# B&R Automation Studio project AcpTrakDemoTemplate (part 2)

#### Main.st
```iecst
(*********************************************************************************
 * Copyright: 	B&R Industrial Automation GmbH
 * Author:    	B&R ES
 * Created:   	April 8, 2022/10:54 AM
 * Description:	All the shuttles crossing this process point will be unsynched.
 * Mandatory: 	NO
 *********************************************************************************)
PROGRAM _INIT

	(*******************************************************************)
	(******************* Process Configuration *************************)
	(*******************************************************************)
	PPAdr 	:= ADR(PP_Test); 	// <-- NAME A VALID PROCESS POINT
	(*** Define in/out speed & acceleration for this process ***)
	// OUT
	Speed_OUT ACCESS ADR(gSpeedEmpty); 	// <-- Bind it to Empty / Full speed global variable
	Acc_OUT	ACCESS ADR(gAccEmpty); 		// <-- Bind it to Empty / Full acceleration global variable
	(*** SceneViewer - Shuttle color after process ***)
	Red	  := 1.0;
	Green := 1.0;
	Blue  := 1.0;
	(********************************************************************)

	(* Local variable to enable/disable the process *)
	CmdEnableProcess := TRUE;
	(* Processpointreference for Functionblocks *)
	MC_BR_TrgPointEnable_AcpTrak_0.ProcessPoint 	:= PPAdr; // <-- NAME A VALID PROCESS POINT
	MC_BR_TrgPointGetInfo_AcpTrak_0.ProcessPoint 	:= PPAdr;	// <-- NAME A VALID PROCESS POINT

END_PROGRAM

PROGRAM _CYCLIC

	//////////////////// HIGH PRIORITY ///////////////////
	IF gTrakAsm.StatusDisabled THEN
		Step 		:= CHECK_TRIGGER;
	END_IF
	//////////////////////////////////////////////////////

	CASE Step OF

		CHECK_TRIGGER:

			(* When the process is enabled and the assembly is ready, the process will be activated *)
			IF((CmdEnableProcess) AND (gTrakAsm.StatusReady))THEN
				MC_BR_TrgPointEnable_AcpTrak_0.Enable := TRUE;
				(* If a shuttle passes the triggerpoint then get the axis reference *)
				IF((MC_BR_TrgPointEnable_AcpTrak_0.Valid) AND (MC_BR_TrgPointEnable_AcpTrak_0.EventCount > 0))THEN
					MC_BR_TrgPointGetInfo_AcpTrak_0.Execute := TRUE;
				END_IF
			ELSE
				(* Else the processpoint will be disabled *)
				MC_BR_TrgPointEnable_AcpTrak_0.Enable := FALSE;
			END_IF

			(* If axis reference is available, save it and go to the next step *)
			IF EDGEPOS(MC_BR_TrgPointGetInfo_AcpTrak_0.Done) THEN
			(* Save axis reference in local variable for use in step machine *)
				ShuttleAxis	:= MC_BR_TrgPointGetInfo_AcpTrak_0.TrgPointInfo.Axis;
				Step 		:= GET_USERDATA;
			END_IF

		GET_USERDATA:

			(* The userdata is copied on a local variable *)
			MC_BR_ShCopyUserData_AcpTrak_0.Axis 		:= ADR(ShuttleAxis);
			MC_BR_ShCopyUserData_AcpTrak_0.Execute 		:= TRUE;
			MC_BR_ShCopyUserData_AcpTrak_0.DataAddress	:= ADR(ShuttleUserData);
			MC_BR_ShCopyUserData_AcpTrak_0.DataSize 	:= SIZEOF(ShuttleUserData);
			MC_BR_ShCopyUserData_AcpTrak_0.Mode 		:= mcACPTRAK_USERDATA_GET;
			(* After copying go to the next step *)
			IF EDGEPOS(MC_BR_ShCopyUserData_AcpTrak_0.Done) THEN
				IF ShuttleUserData.InitDone THEN
					Step := SET_USERDATA;
				ELSE
					Step := CHECK_TRIGGER;
				END_IF
			END_IF

		SET_USERDATA:

			(* Change color to know that shuttles are in unsync. *)
			ShuttleUserData.SceneColorRed 	:= Red;
			ShuttleUserData.SceneColorGreen := Green;
			ShuttleUserData.SceneColorBlue	:= Blue;

			(* The modified userdata will be copied back on the shuttle *)
			MC_BR_ShCopyUserData_AcpTrak_0.Axis 		:= ADR(ShuttleAxis);
			MC_BR_ShCopyUserData_AcpTrak_0.Execute 		:= TRUE;
			MC_BR_ShCopyUserData_AcpTrak_0.DataAddress	:= ADR(ShuttleUserData);
			MC_BR_ShCopyUserData_AcpTrak_0.DataSize 	:= SIZEOF(ShuttleUserData);
			MC_BR_ShCopyUserData_AcpTrak_0.Mode 		:= mcACPTRAK_USERDATA_SET;
			Step := SET_USERDATA_WAIT;

		SET_USERDATA_WAIT:

			IF (MC_BR_ShCopyUserData_AcpTrak_0.Done) THEN
				Step := GO_TO_NEXT_STATION;
			END_IF

		GO_TO_NEXT_STATION:

			MC_BR_ElasticMoveVel_AcpTrak_0.Axis 	:= ADR(ShuttleAxis);
			MC_BR_ElasticMoveVel_AcpTrak_0.Execute	:= TRUE;

			Step := CHECK_TRIGGER;

	END_CASE

	(*** Call all function blocks ***)
	// MC_BR_TrgPointEnable_AcpTrak
	MC_BR_TrgPointEnable_AcpTrak_0();
	// MC_BR_TrgPointGetInfo_AcpTrak
	MC_BR_TrgPointGetInfo_AcpTrak_0();
	MC_BR_TrgPointGetInfo_AcpTrak_0.Execute  := FALSE;
	// MC_BR_ShCopyUserData_AcpTrak
	MC_BR_ShCopyUserData_AcpTrak_0();
	MC_BR_ShCopyUserData_AcpTrak_0.Execute 	 := FALSE;
	//MC_BR_ElasticMoveVel_AcpTrak_0
	MC_BR_ElasticMoveVel_AcpTrak_0.Velocity		:= Speed_OUT;
	MC_BR_ElasticMoveVel_AcpTrak_0.Acceleration	:= Acc_OUT;
	MC_BR_ElasticMoveVel_AcpTrak_0.Deceleration	:= Acc_OUT;
	MC_BR_ElasticMoveVel_AcpTrak_0.Direction	:= mcDIR_POSITIVE;
	MC_BR_ElasticMoveVel_AcpTrak_0();
	MC_BR_ElasticMoveVel_AcpTrak_0.Execute		:= FALSE;

END_PROGRAM
```

### Program Logical/Source/ProcessTemplate/PairedSh/ProcStop_P1 (IEC) - trak process - 1 pair of shuttles wait predefined time

#### Types.typ
```iecst
(*enum*)

TYPE
	StepEnum :
		(
		CHECK_TRIGGER,
		GET_SHUTTLE_DATA,
		GET_SHUTTLE_DATA_WAIT,
		GO_TO_PROCESS_STATION,
		GO_TO_PROCESS_STATION_WAIT,
		WAIT,
		SET_SHUTTLE_DATA,
		SET_SHUTTLE_DATA_WAIT,
		GO_TO_NEXT_STATION
		);
END_TYPE
```

#### Variables.var
```iecst
(*process configuration*)
VAR
	PPAdr : UDINT;
	SecAdr : UDINT;
END_VAR
(*commands*)
VAR
	CmdEnableProcess : BOOL;
END_VAR
(*sequence control*)
VAR
	Step : StepEnum;
	ShuttleAxis : ARRAY[1..2] OF McAxisType;
	ShuttleUserData : ARRAY[1..2] OF TrakShuttleUserDataType;
	WaitTime : UDINT := 500;
	ProcPointPos : LREAL;
	CntShuttle : USINT;
	ReleaseSts : BOOL;
END_VAR
(*colour configuration*)
VAR
	Red : REAL;
	Green : REAL;
	Blue : REAL;
END_VAR
(*movement configuration*)
VAR
	Speed_IN : REFERENCE TO REAL;
	Acc_IN : REFERENCE TO REAL;
	Speed_OUT : REFERENCE TO REAL;
	Acc_OUT : REFERENCE TO REAL;
END_VAR
(*FUB*)
VAR
	MC_BR_AsmReadStatus_AcpTrak_0 : MC_BR_AsmReadStatus_AcpTrak;
	MC_BR_TrgPointEnable_AcpTrak_0 : MC_BR_TrgPointEnable_AcpTrak;
	MC_BR_TrgPointGetInfo_AcpTrak_0 : MC_BR_TrgPointGetInfo_AcpTrak;
	MC_BR_ShCopyUserData_AcpTrak_0 : MC_BR_ShCopyUserData_AcpTrak;
	MC_BR_RoutedMoveAbs_AcpTrak_0 : MC_BR_RoutedMoveAbs_AcpTrak;
	MC_BR_ElasticMoveVel_AcpTrak_0 : MC_BR_ElasticMoveVel_AcpTrak;
	MC_BR_ProcPointGetInfo_AcpTrak_0 : MC_BR_ProcPointGetInfo_AcpTrak;
	TON_0 : TON;
END_VAR
```

#### Main.st
```iecst
(*********************************************************************************
 * Copyright: 	B&R Industrial Automation GmbH
 * Author:    	B&R ES
 * Created:   	April 8, 2022/10:54 AM
 * Description:	One pair of coupled shuttles will be stopped a predefined time in the
				process	station.
 * Mandatory: 	NO
 *********************************************************************************)
PROGRAM _INIT

	(*******************************************************************)
	(******************* Process Configuration *************************)
	(*******************************************************************)
	PPAdr 	:= ADR(PP_Test); 		// <-- NAME A VALID PROCESS POINT
	SecAdr	:= ADR(SectorTrackA);	// <-- NAME A VALID SECTOR
	(*** Define in/out speed & acceleration for this process ***)
	// IN
	Speed_IN ACCESS	ADR(gSpeedEmpty); 	// <-- Bind it to Empty / Full speed global variable
	Acc_IN ACCESS ADR(gAccEmpty); 		// <-- Bind it to Empty / Full acceleration global variable
	// OUT
	Speed_OUT ACCESS ADR(gSpeedFull); 	// <-- Bind it to Empty / Full speed global variable
	Acc_OUT	ACCESS ADR(gAccFull); 		// <-- Bind it to Empty / Full acceleration global variable
	(*** Define Wait Time (ms) ***)
	WaitTime := 500;
	(*** Define if it is a release station ***)
	ReleaseSts := FALSE;
	(*** SceneViewer - Shuttle color after process ***)
	Red	  := 0.02;
	Green := 0.77;
	Blue  := 0.21;
	(********************************************************************)

	CmdEnableProcess 	:= TRUE;
	Step 				:= CHECK_TRIGGER;

	MC_BR_ProcPointGetInfo_AcpTrak_0.ProcessPoint   := PPAdr;
	MC_BR_ProcPointGetInfo_AcpTrak_0.Execute		:= TRUE;

	REPEAT
		MC_BR_ProcPointGetInfo_AcpTrak_0();
	UNTIL
		MC_BR_ProcPointGetInfo_AcpTrak_0.Done OR MC_BR_ProcPointGetInfo_AcpTrak_0.Error
	END_REPEAT;

	ProcPointPos 	:= MC_BR_ProcPointGetInfo_AcpTrak_0.ProcPointInfo.SectorPosition.Position;
	CntShuttle 		:= 1;

END_PROGRAM

PROGRAM _CYCLIC

	///////////////// HIGH PRIORITY /////////////////
	(* reset process sequence if assembly is disabled *)
	IF EDGEPOS(gTrakAsm.StatusDisabled) THEN
		CntShuttle 		:= 1;
		TON_0.IN		:= FALSE;
		Step 			:= CHECK_TRIGGER;
	END_IF

	(***********************************************************************)
	(************************* STATE MACHINE *******************************)
	(***********************************************************************)

	CASE Step OF

		(* enable trigger and wait for one shuttle to pass *)
		CHECK_TRIGGER:
			IF((CmdEnableProcess) AND (MC_BR_AsmReadStatus_AcpTrak_0.AssemblyReady))THEN
				MC_BR_TrgPointEnable_AcpTrak_0.ProcessPoint  := PPAdr;
				MC_BR_TrgPointEnable_AcpTrak_0.Enable        := TRUE;
				(* shuttle passed => get axis reference *)
				IF((MC_BR_TrgPointEnable_AcpTrak_0.Valid) AND (MC_BR_TrgPointEnable_AcpTrak_0.EventCount > 0))THEN
					MC_BR_TrgPointGetInfo_AcpTrak_0.ProcessPoint  := PPAdr;
					MC_BR_TrgPointGetInfo_AcpTrak_0.Execute       := TRUE;
					Step := GET_SHUTTLE_DATA;
				END_IF
			ELSE
				MC_BR_TrgPointEnable_AcpTrak_0.Enable  := FALSE;
			END_IF

		(* axis reference of passed shuttle available *)
		(* get shuttle-UserData *)
		GET_SHUTTLE_DATA:

			IF(MC_BR_TrgPointGetInfo_AcpTrak_0.Done)THEN
				ShuttleAxis[CntShuttle] := MC_BR_TrgPointGetInfo_AcpTrak_0.TrgPointInfo.Axis;
				// read UserData from shuttle
				MC_BR_ShCopyUserData_AcpTrak_0.Axis         := ADR(ShuttleAxis[CntShuttle]);
				MC_BR_ShCopyUserData_AcpTrak_0.Execute      := TRUE;
				MC_BR_ShCopyUserData_AcpTrak_0.DataAddress  := ADR(ShuttleUserData[CntShuttle]);
				MC_BR_ShCopyUserData_AcpTrak_0.DataSize     := SIZEOF(ShuttleUserData[CntShuttle]);
				MC_BR_ShCopyUserData_AcpTrak_0.Mode         := mcACPTRAK_USERDATA_GET;
				Step := GET_SHUTTLE_DATA_WAIT;
			END_IF

		(* wait for shuttle-UserData content available *)
		GET_SHUTTLE_DATA_WAIT:
			IF(MC_BR_ShCopyUserData_AcpTrak_0.Done)THEN
				IF ShuttleUserData[CntShuttle].InitDone THEN
					CASE CntShuttle OF
						// Master
						1:
							Step := GO_TO_PROCESS_STATION;
						// Slave
						2:
							Step := SET_SHUTTLE_DATA;
					END_CASE
				ELSE
					Step := CHECK_TRIGGER;
				END_IF
			END_IF

		GO_TO_PROCESS_STATION:

			MC_BR_RoutedMoveAbs_AcpTrak_0.Axis			:= ADR(ShuttleAxis[CntShuttle]);
			MC_BR_RoutedMoveAbs_AcpTrak_0.Position 		:= ProcPointPos + (gProductWidth/2);
			MC_BR_RoutedMoveAbs_AcpTrak_0.Execute 		:= TRUE;

			CntShuttle 	:= CntShuttle + 1;
			Step 		:= GO_TO_PROCESS_STATION_WAIT;

		GO_TO_PROCESS_STATION_WAIT:

			IF (MC_BR_RoutedMoveAbs_AcpTrak_0.Done) THEN
				TON_0.IN 	:= TRUE;
				Step 		:= WAIT;
			END_IF

		WAIT:

			IF TON_0.Q THEN
				TON_0.IN 	:= FALSE;
				CntShuttle 	:= 1;
				Step 		:= SET_SHUTTLE_DATA;
			END_IF

		(* write modified UserData back to shuttle *)
		SET_SHUTTLE_DATA:

			ShuttleUserData[CntShuttle].SceneColorRed	:= Red;
			ShuttleUserData[CntShuttle].SceneColorGreen	:= Green;
			ShuttleUserData[CntShuttle].SceneColorBlue 	:= Blue;

			MC_BR_ShCopyUserData_AcpTrak_0.Axis         := ADR(ShuttleAxis[CntShuttle]);
			MC_BR_ShCopyUserData_AcpTrak_0.Execute      := TRUE;
			MC_BR_ShCopyUserData_AcpTrak_0.DataAddress  := ADR(ShuttleUserData[CntShuttle]);
			MC_BR_ShCopyUserData_AcpTrak_0.DataSize     := SIZEOF(ShuttleUserData[CntShuttle]);
			MC_BR_ShCopyUserData_AcpTrak_0.Mode         := mcACPTRAK_USERDATA_SET;
			Step := SET_SHUTTLE_DATA_WAIT;

		(* wait for shuttle-UserData content set *)
		SET_SHUTTLE_DATA_WAIT:
			IF(MC_BR_ShCopyUserData_AcpTrak_0.Done)THEN

				CASE CntShuttle OF
					1:
						CntShuttle 	:= CntShuttle + 1;
						Step		:= GO_TO_NEXT_STATION;
					2:
						CntShuttle	:= 1;
						Step 		:= CHECK_TRIGGER;
				END_CASE

			END_IF

			(* go to next station *)
		GO_TO_NEXT_STATION:

			MC_BR_ElasticMoveVel_AcpTrak_0.Axis           := ADR(ShuttleAxis[1]);
			MC_BR_ElasticMoveVel_AcpTrak_0.Execute        := TRUE;

			IF ReleaseSts THEN
				gProducedProduct := gProducedProduct + 1;
			END_IF

			Step := CHECK_TRIGGER;

	END_CASE

	(*** Call all function blocks ***)
	// MC_BR_AsmReadStatus_AcpTrak
	MC_BR_AsmReadStatus_AcpTrak_0.Assembly 	:= ADR(gAssembly_1);
	MC_BR_AsmReadStatus_AcpTrak_0.Enable 	:= TRUE;
	MC_BR_AsmReadStatus_AcpTrak_0();
    // MC_BR_TrgPointEnable_AcpTrak
	MC_BR_TrgPointEnable_AcpTrak_0();
    // MC_BR_TrgPointGetInfo_AcpTrak
	MC_BR_TrgPointGetInfo_AcpTrak_0();
	MC_BR_TrgPointGetInfo_AcpTrak_0.Execute := FALSE;
    // TON_0
	TON_0.PT := UDINT_TO_TIME(WaitTime);
	TON_0();
	// MC_BR_ShCopyUserData_AcpTrak
	MC_BR_ShCopyUserData_AcpTrak_0();
	MC_BR_ShCopyUserData_AcpTrak_0.Execute := FALSE;
	// MC_BR_RoutedMoveAbs_AcpTrak_0
	MC_BR_RoutedMoveAbs_AcpTrak_0.Sector 		  := SecAdr;
	MC_BR_RoutedMoveAbs_AcpTrak_0.Velocity		  := Speed_IN;
	MC_BR_RoutedMoveAbs_AcpTrak_0.Acceleration	  := Acc_IN;
	MC_BR_RoutedMoveAbs_AcpTrak_0.Deceleration	  := Acc_IN;
	MC_BR_RoutedMoveAbs_AcpTrak_0();
	MC_BR_RoutedMoveAbs_AcpTrak_0.Execute := FALSE;
	// MC_BR_ElasticMoveVel_AcpTrak_0
	MC_BR_ElasticMoveVel_AcpTrak_0.Velocity       := Speed_OUT;
	MC_BR_ElasticMoveVel_AcpTrak_0.Acceleration   := Acc_OUT;
	MC_BR_ElasticMoveVel_AcpTrak_0.Deceleration   := Acc_OUT;
	MC_BR_ElasticMoveVel_AcpTrak_0.Jerk           := 0.0;
	MC_BR_ElasticMoveVel_AcpTrak_0.Direction	  := mcDIR_POSITIVE;
	MC_BR_ElasticMoveVel_AcpTrak_0.BufferMode     := mcABORTING;
	MC_BR_ElasticMoveVel_AcpTrak_0();
	MC_BR_ElasticMoveVel_AcpTrak_0.Execute := FALSE;

END_PROGRAM
```

### Program Logical/Source/ProcessTemplate/PairedSh/ProcStop_P2 (IEC) - trak process - 2 pair of shuttles wait predefined time

#### Types.typ
```iecst
(*enum*)

TYPE
	StepEnum :
		(
		CHECK_TRIGGER,
		GET_SHUTTLE_DATA,
		GET_SHUTTLE_DATA_WAIT,
		GO_TO_PROCESS_STATION_1,
		GO_TO_PROCESS_STATION_2,
		GO_TO_PROCESS_STATION_WAIT,
		WAIT,
		SET_SHUTTLE_DATA,
		SET_SHUTTLE_DATA_WAIT,
		GO_TO_NEXT_STATION
		);
END_TYPE
```

#### Variables.var
```iecst
(*process configuration*)
VAR
	PPAdr : UDINT;
	SecAdr : UDINT;
END_VAR
(*commands*)
VAR
	CmdEnableProcess : BOOL;
END_VAR
(*sequence control*)
VAR
	Step : StepEnum;
	ShuttleAxis : ARRAY[1..4] OF McAxisType;
	ShuttleUserData : ARRAY[1..4] OF TrakShuttleUserDataType;
	WaitTime : UDINT := 500;
	ProcPointPos : LREAL;
	CntShuttle : USINT;
	DistTravelled : LREAL;
	ReleaseSts : BOOL;
END_VAR
(*colour configuration*)
VAR
	Red : REAL;
	Green : REAL;
	Blue : REAL;
END_VAR
(*movement configuration*)
VAR
	Speed_IN : REFERENCE TO REAL;
	Acc_IN : REFERENCE TO REAL;
	Speed_OUT : REFERENCE TO REAL;
	Acc_OUT : REFERENCE TO REAL;
END_VAR
(*FUB*)
VAR
	MC_BR_AsmReadStatus_AcpTrak_0 : MC_BR_AsmReadStatus_AcpTrak;
	MC_BR_TrgPointEnable_AcpTrak_0 : MC_BR_TrgPointEnable_AcpTrak;
	MC_BR_TrgPointGetInfo_AcpTrak_0 : MC_BR_TrgPointGetInfo_AcpTrak;
	MC_BR_ShCopyUserData_AcpTrak_0 : MC_BR_ShCopyUserData_AcpTrak;
	MC_BR_RoutedMoveAbs_AcpTrak_0 : MC_BR_RoutedMoveAbs_AcpTrak;
	MC_BR_RoutedMoveAbs_AcpTrak_1 : MC_BR_RoutedMoveAbs_AcpTrak;
	MC_BR_ElasticMoveVel_AcpTrak_0 : MC_BR_ElasticMoveVel_AcpTrak;
	MC_BR_ElasticMoveVel_AcpTrak_1 : MC_BR_ElasticMoveVel_AcpTrak;
	MC_BR_ProcPointGetInfo_AcpTrak_0 : MC_BR_ProcPointGetInfo_AcpTrak;
	MC_ReadStatus_0 : MC_ReadStatus;
	MC_ReadStatus_1 : MC_ReadStatus;
	TON_0 : TON;
END_VAR
```

#### Main.st
```iecst
(*********************************************************************************
 * Copyright: 	B&R Industrial Automation GmbH
 * Author:    	B&R ES
 * Created:   	April 8, 2022/10:54 AM
 * Description:	Two pairs of coupled shuttles will be stopped a predefined time in the
				process	station.
 * Mandatory: 	NO
 *********************************************************************************)
PROGRAM _INIT

	(*******************************************************************)
	(******************* Process Configuration *************************)
	(*******************************************************************)
	PPAdr 	:= ADR(PP_Test); 		// <-- NAME A VALID PROCESS POINT
	SecAdr	:= ADR(SectorTrackA);	// <-- NAME A VALID SECTOR
	(*** Define in/out speed & acceleration for this process ***)
	// IN
	Speed_IN ACCESS	ADR(gSpeedEmpty); 	// <-- Bind it to Empty / Full speed global variable
	Acc_IN ACCESS ADR(gAccEmpty); 		// <-- Bind it to Empty / Full acceleration global variable
	// OUT
	Speed_OUT ACCESS ADR(gSpeedFull); 	// <-- Bind it to Empty / Full speed global variable
	Acc_OUT	ACCESS ADR(gAccFull); 		// <-- Bind it to Empty / Full acceleration global variable
	(*** Define Wait Time (ms) ***)
	WaitTime := 500;
	(*** Define relative center point distance for the first coupled shuttles ***)
	DistTravelled	:= 0.33;
	(*** Define if it is a release station ***)
	ReleaseSts := FALSE;
	(*** SceneViewer - Shuttle color after process ***)
	Red	  := 0.02;
	Green := 0.77;
	Blue  := 0.21;
	(********************************************************************)

	CmdEnableProcess 	:= TRUE;
	Step 				:= CHECK_TRIGGER;

	MC_BR_ProcPointGetInfo_AcpTrak_0.ProcessPoint   := PPAdr;
	MC_BR_ProcPointGetInfo_AcpTrak_0.Execute		:= TRUE;

	REPEAT
		MC_BR_ProcPointGetInfo_AcpTrak_0();
	UNTIL
		MC_BR_ProcPointGetInfo_AcpTrak_0.Done OR MC_BR_ProcPointGetInfo_AcpTrak_0.Error
	END_REPEAT;

	ProcPointPos 	:= MC_BR_ProcPointGetInfo_AcpTrak_0.ProcPointInfo.SectorPosition.Position;
	CntShuttle 		:= 1;

END_PROGRAM

PROGRAM _CYCLIC

	///////////////// HIGH PRIORITY /////////////////
	(* reset process sequence if assembly is disabled *)
	IF EDGEPOS(gTrakAsm.StatusDisabled) THEN
		CntShuttle 		:= 1;
		TON_0.IN		:= FALSE;
		Step 			:= CHECK_TRIGGER;
	END_IF

	(***********************************************************************)
	(************************* STATE MACHINE *******************************)
	(***********************************************************************)

	CASE Step OF

		(* enable trigger and wait for one shuttle to pass *)
		CHECK_TRIGGER:
			IF((CmdEnableProcess) AND (MC_BR_AsmReadStatus_AcpTrak_0.AssemblyReady))THEN
				MC_BR_TrgPointEnable_AcpTrak_0.ProcessPoint  := PPAdr;
				MC_BR_TrgPointEnable_AcpTrak_0.Enable        := TRUE;
				(* shuttle passed => get axis reference *)
				IF((MC_BR_TrgPointEnable_AcpTrak_0.Valid) AND (MC_BR_TrgPointEnable_AcpTrak_0.EventCount > 0))THEN
					MC_BR_TrgPointGetInfo_AcpTrak_0.ProcessPoint  := PPAdr;
					MC_BR_TrgPointGetInfo_AcpTrak_0.Execute       := TRUE;
					Step := GET_SHUTTLE_DATA;
				END_IF
			ELSE
				MC_BR_TrgPointEnable_AcpTrak_0.Enable  := FALSE;
			END_IF

			(* axis reference of passed shuttle available *)
			(* get shuttle-UserData *)
		GET_SHUTTLE_DATA:

			IF(MC_BR_TrgPointGetInfo_AcpTrak_0.Done)THEN
				ShuttleAxis[CntShuttle] := MC_BR_TrgPointGetInfo_AcpTrak_0.TrgPointInfo.Axis;
				// read UserData from shuttle
				MC_BR_ShCopyUserData_AcpTrak_0.Axis         := ADR(ShuttleAxis[CntShuttle]);
				MC_BR_ShCopyUserData_AcpTrak_0.Execute      := TRUE;
				MC_BR_ShCopyUserData_AcpTrak_0.DataAddress  := ADR(ShuttleUserData[CntShuttle]);
				MC_BR_ShCopyUserData_AcpTrak_0.DataSize     := SIZEOF(ShuttleUserData[CntShuttle]);
				MC_BR_ShCopyUserData_AcpTrak_0.Mode         := mcACPTRAK_USERDATA_GET;
				Step := GET_SHUTTLE_DATA_WAIT;
			END_IF

			(* wait for shuttle-UserData content available *)
		GET_SHUTTLE_DATA_WAIT:
			IF(MC_BR_ShCopyUserData_AcpTrak_0.Done)THEN
				IF ShuttleUserData[CntShuttle].InitDone THEN
					CASE CntShuttle OF
						// Master from first pair
						1:
							Step := GO_TO_PROCESS_STATION_1;
						// Slave from first pair
						2:
							CntShuttle 	:= CntShuttle + 1;
							Step 		:= CHECK_TRIGGER;
						// Master from second pair
						3:
							Step := GO_TO_PROCESS_STATION_2;
						// Slave from second pair
						4:
							Step := SET_SHUTTLE_DATA;
					END_CASE
				ELSE
					Step := CHECK_TRIGGER;
				END_IF
			END_IF

		GO_TO_PROCESS_STATION_1:

			MC_BR_RoutedMoveAbs_AcpTrak_0.Axis			:= ADR(ShuttleAxis[CntShuttle]);
			MC_BR_RoutedMoveAbs_AcpTrak_0.Position 		:= ProcPointPos + (gProductWidth/2) + DistTravelled;
			MC_BR_RoutedMoveAbs_AcpTrak_0.Execute 		:= TRUE;

			CntShuttle 	:= CntShuttle + 1;
			Step 		:= CHECK_TRIGGER;

		GO_TO_PROCESS_STATION_2:

			MC_BR_RoutedMoveAbs_AcpTrak_1.Axis		:= ADR(ShuttleAxis[CntShuttle]);
			MC_BR_RoutedMoveAbs_AcpTrak_1.Position 	:= ProcPointPos + (gProductWidth/2);
			MC_BR_RoutedMoveAbs_AcpTrak_1.Execute 	:= TRUE;

			Step := GO_TO_PROCESS_STATION_WAIT;

		GO_TO_PROCESS_STATION_WAIT:

			MC_ReadStatus_0.Axis 	:= ADR(ShuttleAxis[1]);
			MC_ReadStatus_0.Enable	:= TRUE;

			MC_ReadStatus_1.Axis 	:= ADR(ShuttleAxis[3]);
			MC_ReadStatus_1.Enable	:= TRUE;

			IF (MC_ReadStatus_0.StandStill AND MC_ReadStatus_1.StandStill) THEN
				MC_ReadStatus_0.Enable := FALSE;
				MC_ReadStatus_1.Enable := FALSE;
				TON_0.IN 	:= TRUE;
				Step 		:= WAIT;
			END_IF

		WAIT:

			IF TON_0.Q THEN
				TON_0.IN 	:= FALSE;
				CntShuttle 	:= 1;
				Step 		:= SET_SHUTTLE_DATA;
			END_IF

		(* write modified UserData back to shuttle *)
		SET_SHUTTLE_DATA:

			ShuttleUserData[CntShuttle].SceneColorRed	:= Red;
			ShuttleUserData[CntShuttle].SceneColorGreen	:= Green;
			ShuttleUserData[CntShuttle].SceneColorBlue 	:= Blue;

			MC_BR_ShCopyUserData_AcpTrak_0.Axis         := ADR(ShuttleAxis[CntShuttle]);
			MC_BR_ShCopyUserData_AcpTrak_0.Execute      := TRUE;
			MC_BR_ShCopyUserData_AcpTrak_0.DataAddress  := ADR(ShuttleUserData[CntShuttle]);
			MC_BR_ShCopyUserData_AcpTrak_0.DataSize     := SIZEOF(ShuttleUserData[CntShuttle]);
			MC_BR_ShCopyUserData_AcpTrak_0.Mode         := mcACPTRAK_USERDATA_SET;
			Step := SET_SHUTTLE_DATA_WAIT;

		(* wait for shuttle-UserData content set *)
		SET_SHUTTLE_DATA_WAIT:
			IF(MC_BR_ShCopyUserData_AcpTrak_0.Done)THEN

				CASE CntShuttle OF
					1..2:
						CntShuttle 	:= CntShuttle + 1;
						Step		:= SET_SHUTTLE_DATA;
					3:
						CntShuttle	:= CntShuttle + 1;
						Step 		:= GO_TO_NEXT_STATION;
					4:
						CntShuttle 	:= 1;
						Step	 	:= CHECK_TRIGGER;
				END_CASE

			END_IF

			(* go to next station *)
		GO_TO_NEXT_STATION:

			MC_BR_ElasticMoveVel_AcpTrak_0.Axis           := ADR(ShuttleAxis[1]);
			MC_BR_ElasticMoveVel_AcpTrak_0.Execute        := TRUE;

			MC_BR_ElasticMoveVel_AcpTrak_1.Axis           := ADR(ShuttleAxis[3]);
			MC_BR_ElasticMoveVel_AcpTrak_1.Execute        := TRUE;

			IF ReleaseSts THEN
				gProducedProduct := gProducedProduct + 2;
			END_IF

			Step := CHECK_TRIGGER;

	END_CASE

	(*** Call all function blocks ***)
	// MC_BR_AsmReadStatus_AcpTrak
	MC_BR_AsmReadStatus_AcpTrak_0.Assembly 	:= ADR(gAssembly_1);
	MC_BR_AsmReadStatus_AcpTrak_0.Enable 	:= TRUE;
	MC_BR_AsmReadStatus_AcpTrak_0();
    // MC_BR_TrgPointEnable_AcpTrak
	MC_BR_TrgPointEnable_AcpTrak_0();
    // MC_BR_TrgPointGetInfo_AcpTrak
	MC_BR_TrgPointGetInfo_AcpTrak_0();
	MC_BR_TrgPointGetInfo_AcpTrak_0.Execute := FALSE;
    // TON_0
	TON_0.PT := UDINT_TO_TIME(WaitTime);
	TON_0();
	// MC_BR_ShCopyUserData_AcpTrak
	MC_BR_ShCopyUserData_AcpTrak_0();
	MC_BR_ShCopyUserData_AcpTrak_0.Execute := FALSE;
	// MC_BR_RoutedMoveAbs_AcpTrak_0
	MC_BR_RoutedMoveAbs_AcpTrak_0.Sector 		  := SecAdr;
	MC_BR_RoutedMoveAbs_AcpTrak_0.Velocity		  := Speed_IN;
	MC_BR_RoutedMoveAbs_AcpTrak_0.Acceleration	  := Acc_IN;
	MC_BR_RoutedMoveAbs_AcpTrak_0.Deceleration	  := Acc_IN;
	MC_BR_RoutedMoveAbs_AcpTrak_0();
	MC_BR_RoutedMoveAbs_AcpTrak_0.Execute := FALSE;
	// MC_BR_RoutedMoveAbs_AcpTrak_1
	MC_BR_RoutedMoveAbs_AcpTrak_1.Sector 		  := SecAdr;
	MC_BR_RoutedMoveAbs_AcpTrak_1.Velocity		  := Speed_IN;
	MC_BR_RoutedMoveAbs_AcpTrak_1.Acceleration	  := Acc_IN;
	MC_BR_RoutedMoveAbs_AcpTrak_1.Deceleration	  := Acc_IN;
	MC_BR_RoutedMoveAbs_AcpTrak_1();
	MC_BR_RoutedMoveAbs_AcpTrak_1.Execute := FALSE;
	// MC_BR_ElasticMoveVel_AcpTrak_0
	MC_BR_ElasticMoveVel_AcpTrak_0.Velocity       := Speed_OUT;
	MC_BR_ElasticMoveVel_AcpTrak_0.Acceleration   := Acc_OUT;
	MC_BR_ElasticMoveVel_AcpTrak_0.Deceleration   := Acc_OUT;
	MC_BR_ElasticMoveVel_AcpTrak_0.Jerk           := 0.0;
	MC_BR_ElasticMoveVel_AcpTrak_0.Direction	  := mcDIR_POSITIVE;
	MC_BR_ElasticMoveVel_AcpTrak_0.BufferMode     := mcABORTING;
	MC_BR_ElasticMoveVel_AcpTrak_0();
	MC_BR_ElasticMoveVel_AcpTrak_0.Execute := FALSE;
	// MC_BR_ElasticMoveVel_AcpTrak_1
	MC_BR_ElasticMoveVel_AcpTrak_1.Velocity       := Speed_OUT;
	MC_BR_ElasticMoveVel_AcpTrak_1.Acceleration   := Acc_OUT;
	MC_BR_ElasticMoveVel_AcpTrak_1.Deceleration   := Acc_OUT;
	MC_BR_ElasticMoveVel_AcpTrak_1.Jerk           := 0.0;
	MC_BR_ElasticMoveVel_AcpTrak_1.Direction	  := mcDIR_POSITIVE;
	MC_BR_ElasticMoveVel_AcpTrak_1.BufferMode     := mcABORTING;
	MC_BR_ElasticMoveVel_AcpTrak_1();
	MC_BR_ElasticMoveVel_AcpTrak_1.Execute := FALSE;
	// MC_ReadStatus
	MC_ReadStatus_0();
	MC_ReadStatus_1();

END_PROGRAM
```

### Program Logical/Source/ProcessTemplate/PairedSh/ProcStop_P3 (IEC) - trak process - 3 pair of shuttles wait predefined time

#### Types.typ
```iecst
(*enum*)

TYPE
	StepEnum :
		(
		CHECK_TRIGGER,
		GET_SHUTTLE_DATA,
		GET_SHUTTLE_DATA_WAIT,
		GO_TO_PROCESS_STATION_1,
		GO_TO_PROCESS_STATION_2,
		GO_TO_PROCESS_STATION_3,
		GO_TO_PROCESS_STATION_WAIT,
		WAIT,
		SET_SHUTTLE_DATA,
		SET_SHUTTLE_DATA_WAIT,
		GO_TO_NEXT_STATION
		);
END_TYPE
```

#### Variables.var
```iecst
(*process configuration*)
VAR
	PPAdr : UDINT;
	SecAdr : UDINT;
END_VAR
(*commands*)
VAR
	CmdEnableProcess : BOOL;
END_VAR
(*sequence control*)
VAR
	Step : StepEnum;
	ShuttleAxis : ARRAY[1..6] OF McAxisType;
	ShuttleUserData : ARRAY[1..6] OF TrakShuttleUserDataType;
	WaitTime : UDINT := 500;
	ProcPointPos : LREAL;
	CntShuttle : USINT;
	DistTravelled_1 : LREAL;
	DistTravelled_2 : LREAL;
	ReleaseSts : BOOL;
END_VAR
(*colour configuration*)
VAR
	Red : REAL;
	Green : REAL;
	Blue : REAL;
END_VAR
(*movement configuration*)
VAR
	Speed_IN : REFERENCE TO REAL;
	Acc_IN : REFERENCE TO REAL;
	Speed_OUT : REFERENCE TO REAL;
	Acc_OUT : REFERENCE TO REAL;
END_VAR
(*FUB*)
VAR
	MC_BR_AsmReadStatus_AcpTrak_0 : MC_BR_AsmReadStatus_AcpTrak;
	MC_BR_TrgPointEnable_AcpTrak_0 : MC_BR_TrgPointEnable_AcpTrak;
	MC_BR_TrgPointGetInfo_AcpTrak_0 : MC_BR_TrgPointGetInfo_AcpTrak;
	MC_BR_ShCopyUserData_AcpTrak_0 : MC_BR_ShCopyUserData_AcpTrak;
	MC_BR_RoutedMoveAbs_AcpTrak_0 : MC_BR_RoutedMoveAbs_AcpTrak;
	MC_BR_RoutedMoveAbs_AcpTrak_1 : MC_BR_RoutedMoveAbs_AcpTrak;
	MC_BR_RoutedMoveAbs_AcpTrak_2 : MC_BR_RoutedMoveAbs_AcpTrak;
	MC_BR_ElasticMoveVel_AcpTrak_0 : MC_BR_ElasticMoveVel_AcpTrak;
	MC_BR_ElasticMoveVel_AcpTrak_1 : MC_BR_ElasticMoveVel_AcpTrak;
	MC_BR_ElasticMoveVel_AcpTrak_2 : MC_BR_ElasticMoveVel_AcpTrak;
	MC_BR_ProcPointGetInfo_AcpTrak_0 : MC_BR_ProcPointGetInfo_AcpTrak;
	MC_ReadStatus_0 : MC_ReadStatus;
	MC_ReadStatus_1 : MC_ReadStatus;
	MC_ReadStatus_2 : MC_ReadStatus;
	TON_0 : TON;
END_VAR
```

#### Main.st
```iecst
(*********************************************************************************
 * Copyright: 	B&R Industrial Automation GmbH
 * Author:    	B&R ES
 * Created:   	April 8, 2022/10:54 AM
 * Description:	Three pairs of coupled shuttles will be stopped a predefined time
				in the process station.
 * Mandatory: 	NO
 *********************************************************************************)
PROGRAM _INIT

	(*******************************************************************)
	(******************* Process Configuration *************************)
	(*******************************************************************)
	PPAdr 	:= ADR(PP_Test); 		// <-- NAME A VALID PROCESS POINT
	SecAdr	:= ADR(SectorTrackA);	// <-- NAME A VALID SECTOR
	(*** Define in/out speed & acceleration for this process ***)
	// IN
	Speed_IN ACCESS	ADR(gSpeedEmpty); 	// <-- Bind it to Empty / Full speed global variable
	Acc_IN ACCESS ADR(gAccEmpty); 		// <-- Bind it to Empty / Full acceleration global variable
	// OUT
	Speed_OUT ACCESS ADR(gSpeedFull); 	// <-- Bind it to Empty / Full speed global variable
	Acc_OUT	ACCESS ADR(gAccFull); 		// <-- Bind it to Empty / Full acceleration global variable
	(*** Define Wait Time (ms) ***)
	WaitTime := 500;
	(*** Define relative center point distance for the first & second coupled shuttles ***)
	DistTravelled_1	:= 0.66;
	DistTravelled_2 := 0.33;
	(*** Define if it is a release station ***)
	ReleaseSts := FALSE;
	(*** SceneViewer - Shuttle color after process ***)
	Red	  := 0.02;
	Green := 0.77;
	Blue  := 0.21;
	(********************************************************************)

	CmdEnableProcess 	:= TRUE;
	Step 				:= CHECK_TRIGGER;

	MC_BR_ProcPointGetInfo_AcpTrak_0.ProcessPoint   := PPAdr;
	MC_BR_ProcPointGetInfo_AcpTrak_0.Execute		:= TRUE;

	REPEAT
		MC_BR_ProcPointGetInfo_AcpTrak_0();
	UNTIL
		MC_BR_ProcPointGetInfo_AcpTrak_0.Done OR MC_BR_ProcPointGetInfo_AcpTrak_0.Error
	END_REPEAT;

	ProcPointPos 	:= MC_BR_ProcPointGetInfo_AcpTrak_0.ProcPointInfo.SectorPosition.Position;
	CntShuttle 		:= 1;

END_PROGRAM

PROGRAM _CYCLIC

	///////////////// HIGH PRIORITY /////////////////
	(* reset process sequence if assembly is disabled *)
	IF EDGEPOS(gTrakAsm.StatusDisabled) THEN
		CntShuttle 		:= 1;
		TON_0.IN		:= FALSE;
		Step 			:= CHECK_TRIGGER;
	END_IF

	(***********************************************************************)
	(************************* STATE MACHINE *******************************)
	(***********************************************************************)

	CASE Step OF

		(* enable trigger and wait for one shuttle to pass *)
		CHECK_TRIGGER:
			IF((CmdEnableProcess) AND (MC_BR_AsmReadStatus_AcpTrak_0.AssemblyReady))THEN
				MC_BR_TrgPointEnable_AcpTrak_0.ProcessPoint  := PPAdr;
				MC_BR_TrgPointEnable_AcpTrak_0.Enable        := TRUE;
				(* shuttle passed => get axis reference *)
				IF((MC_BR_TrgPointEnable_AcpTrak_0.Valid) AND (MC_BR_TrgPointEnable_AcpTrak_0.EventCount > 0))THEN
					MC_BR_TrgPointGetInfo_AcpTrak_0.ProcessPoint  := PPAdr;
					MC_BR_TrgPointGetInfo_AcpTrak_0.Execute       := TRUE;
					Step := GET_SHUTTLE_DATA;
				END_IF
			ELSE
				MC_BR_TrgPointEnable_AcpTrak_0.Enable  := FALSE;
			END_IF

			(* axis reference of passed shuttle available *)
			(* get shuttle-UserData *)
		GET_SHUTTLE_DATA:

			IF(MC_BR_TrgPointGetInfo_AcpTrak_0.Done)THEN
				ShuttleAxis[CntShuttle] := MC_BR_TrgPointGetInfo_AcpTrak_0.TrgPointInfo.Axis;
				// read UserData from shuttle
				MC_BR_ShCopyUserData_AcpTrak_0.Axis         := ADR(ShuttleAxis[CntShuttle]);
				MC_BR_ShCopyUserData_AcpTrak_0.Execute      := TRUE;
				MC_BR_ShCopyUserData_AcpTrak_0.DataAddress  := ADR(ShuttleUserData[CntShuttle]);
				MC_BR_ShCopyUserData_AcpTrak_0.DataSize     := SIZEOF(ShuttleUserData[CntShuttle]);
				MC_BR_ShCopyUserData_AcpTrak_0.Mode         := mcACPTRAK_USERDATA_GET;
				Step := GET_SHUTTLE_DATA_WAIT;
			END_IF

			(* wait for shuttle-UserData content available *)
		GET_SHUTTLE_DATA_WAIT:
			IF(MC_BR_ShCopyUserData_AcpTrak_0.Done)THEN
				IF ShuttleUserData[CntShuttle].InitDone THEN
					CASE CntShuttle OF
						// Master from first pair
						1:
							Step := GO_TO_PROCESS_STATION_1;
						// Slave from first pair
						2:
							CntShuttle 	:= CntShuttle + 1;
							Step 		:= CHECK_TRIGGER;
						// Master from second pair
						3:
							Step := GO_TO_PROCESS_STATION_2;
						// Slave from second pair
						4:
							CntShuttle 	:= CntShuttle + 1;
							Step 		:= CHECK_TRIGGER;
						// Master from third pair
						5:
							Step := GO_TO_PROCESS_STATION_3;
						// Slave from third pair
						6:
							Step := SET_SHUTTLE_DATA;
					END_CASE
				ELSE
					Step := CHECK_TRIGGER;
				END_IF
			END_IF

		GO_TO_PROCESS_STATION_1:

			MC_BR_RoutedMoveAbs_AcpTrak_0.Axis		:= ADR(ShuttleAxis[CntShuttle]);
			MC_BR_RoutedMoveAbs_AcpTrak_0.Position 	:= ProcPointPos + (gProductWidth/2) + DistTravelled_1;
			MC_BR_RoutedMoveAbs_AcpTrak_0.Execute 	:= TRUE;

			CntShuttle 	:= CntShuttle + 1;
			Step 		:= CHECK_TRIGGER;

		GO_TO_PROCESS_STATION_2:

			MC_BR_RoutedMoveAbs_AcpTrak_1.Axis		:= ADR(ShuttleAxis[CntShuttle]);
			MC_BR_RoutedMoveAbs_AcpTrak_1.Position 	:= ProcPointPos + (gProductWidth/2) + DistTravelled_2;
			MC_BR_RoutedMoveAbs_AcpTrak_1.Execute 	:= TRUE;

			CntShuttle 	:= CntShuttle + 1;
			Step 		:= CHECK_TRIGGER;

		GO_TO_PROCESS_STATION_3:

			MC_BR_RoutedMoveAbs_AcpTrak_2.Axis		:= ADR(ShuttleAxis[CntShuttle]);
			MC_BR_RoutedMoveAbs_AcpTrak_2.Position 	:= ProcPointPos + (gProductWidth/2);
			MC_BR_RoutedMoveAbs_AcpTrak_2.Execute 	:= TRUE;

			Step	:= GO_TO_PROCESS_STATION_WAIT;

		GO_TO_PROCESS_STATION_WAIT:

			MC_ReadStatus_0.Axis 	:= ADR(ShuttleAxis[1]);
			MC_ReadStatus_0.Enable	:= TRUE;

			MC_ReadStatus_1.Axis 	:= ADR(ShuttleAxis[3]);
			MC_ReadStatus_1.Enable	:= TRUE;

			MC_ReadStatus_2.Axis 	:= ADR(ShuttleAxis[5]);
			MC_ReadStatus_2.Enable	:= TRUE;

			IF (MC_ReadStatus_0.StandStill AND MC_ReadStatus_1.StandStill AND MC_ReadStatus_2.StandStill) THEN
				MC_ReadStatus_0.Enable := FALSE;
				MC_ReadStatus_1.Enable := FALSE;
				MC_ReadStatus_2.Enable := FALSE;
				TON_0.IN 	:= TRUE;
				Step 		:= WAIT;
			END_IF

		(* dependent of shuttle-UserData content => shuttle will be rerouted on Process Point Check *)
		WAIT:

			IF TON_0.Q THEN
				TON_0.IN 	:= FALSE;
				CntShuttle 	:= 1;
				Step 		:= SET_SHUTTLE_DATA;
			END_IF

		(* write modified UserData back to shuttle *)
		SET_SHUTTLE_DATA:

			ShuttleUserData[CntShuttle].SceneColorRed	:= Red;
			ShuttleUserData[CntShuttle].SceneColorGreen	:= Green;
			ShuttleUserData[CntShuttle].SceneColorBlue 	:= Blue;

			MC_BR_ShCopyUserData_AcpTrak_0.Axis         := ADR(ShuttleAxis[CntShuttle]);
			MC_BR_ShCopyUserData_AcpTrak_0.Execute      := TRUE;
			MC_BR_ShCopyUserData_AcpTrak_0.DataAddress  := ADR(ShuttleUserData[CntShuttle]);
			MC_BR_ShCopyUserData_AcpTrak_0.DataSize     := SIZEOF(ShuttleUserData[CntShuttle]);
			MC_BR_ShCopyUserData_AcpTrak_0.Mode         := mcACPTRAK_USERDATA_SET;
			Step := SET_SHUTTLE_DATA_WAIT;

		(* wait for shuttle-UserData content set *)
		SET_SHUTTLE_DATA_WAIT:
			IF(MC_BR_ShCopyUserData_AcpTrak_0.Done)THEN

				CASE CntShuttle OF
					1..4:
						CntShuttle 	:= CntShuttle + 1;
						Step		:= SET_SHUTTLE_DATA;
					5:
						CntShuttle	:= CntShuttle + 1;
						Step 		:= GO_TO_NEXT_STATION;
					6:
						CntShuttle 	:= 1;
						Step	 	:= CHECK_TRIGGER;

				END_CASE

			END_IF

			(* go to next station *)
		GO_TO_NEXT_STATION:

			MC_BR_ElasticMoveVel_AcpTrak_0.Axis           := ADR(ShuttleAxis[1]);
			MC_BR_ElasticMoveVel_AcpTrak_0.Execute        := TRUE;

			MC_BR_ElasticMoveVel_AcpTrak_1.Axis           := ADR(ShuttleAxis[3]);
			MC_BR_ElasticMoveVel_AcpTrak_1.Execute        := TRUE;

			MC_BR_ElasticMoveVel_AcpTrak_2.Axis           := ADR(ShuttleAxis[5]);
			MC_BR_ElasticMoveVel_AcpTrak_2.Execute        := TRUE;

			IF ReleaseSts THEN
				gProducedProduct := gProducedProduct + 3;
			END_IF

			Step := CHECK_TRIGGER;

	END_CASE

	(*** Call all function blocks ***)
	// MC_BR_AsmReadStatus_AcpTrak
	MC_BR_AsmReadStatus_AcpTrak_0.Assembly 	:= ADR(gAssembly_1);
	MC_BR_AsmReadStatus_AcpTrak_0.Enable 	:= TRUE;
	MC_BR_AsmReadStatus_AcpTrak_0();
    // MC_BR_TrgPointEnable_AcpTrak
	MC_BR_TrgPointEnable_AcpTrak_0();
    // MC_BR_TrgPointGetInfo_AcpTrak
	MC_BR_TrgPointGetInfo_AcpTrak_0();
	MC_BR_TrgPointGetInfo_AcpTrak_0.Execute := FALSE;
    // TON_0
	TON_0.PT := UDINT_TO_TIME(WaitTime);
	TON_0();
	// MC_BR_ShCopyUserData_AcpTrak
	MC_BR_ShCopyUserData_AcpTrak_0();
	MC_BR_ShCopyUserData_AcpTrak_0.Execute := FALSE;
	// MC_BR_RoutedMoveAbs_AcpTrak_0
	MC_BR_RoutedMoveAbs_AcpTrak_0.Sector 		  := SecAdr;
	MC_BR_RoutedMoveAbs_AcpTrak_0.Velocity		  := Speed_IN;
	MC_BR_RoutedMoveAbs_AcpTrak_0.Acceleration	  := Acc_IN;
	MC_BR_RoutedMoveAbs_AcpTrak_0.Deceleration	  := Acc_IN;
	MC_BR_RoutedMoveAbs_AcpTrak_0();
	MC_BR_RoutedMoveAbs_AcpTrak_0.Execute := FALSE;
	// MC_BR_RoutedMoveAbs_AcpTrak_1
	MC_BR_RoutedMoveAbs_AcpTrak_1.Sector 		  := SecAdr;
	MC_BR_RoutedMoveAbs_AcpTrak_1.Velocity		  := Speed_IN;
	MC_BR_RoutedMoveAbs_AcpTrak_1.Acceleration	  := Acc_IN;
	MC_BR_RoutedMoveAbs_AcpTrak_1.Deceleration	  := Acc_IN;
	MC_BR_RoutedMoveAbs_AcpTrak_1();
	MC_BR_RoutedMoveAbs_AcpTrak_1.Execute := FALSE;
	// MC_BR_RoutedMoveAbs_AcpTrak_2
	MC_BR_RoutedMoveAbs_AcpTrak_2.Sector 		  := SecAdr;
	MC_BR_RoutedMoveAbs_AcpTrak_2.Velocity		  := Speed_IN;
	MC_BR_RoutedMoveAbs_AcpTrak_2.Acceleration	  := Acc_IN;
	MC_BR_RoutedMoveAbs_AcpTrak_2.Deceleration	  := Acc_IN;
	MC_BR_RoutedMoveAbs_AcpTrak_2();
	MC_BR_RoutedMoveAbs_AcpTrak_2.Execute := FALSE;
	// MC_BR_ElasticMoveVel_AcpTrak_0
	MC_BR_ElasticMoveVel_AcpTrak_0.Velocity       := Speed_OUT;
	MC_BR_ElasticMoveVel_AcpTrak_0.Acceleration   := Acc_OUT;
	MC_BR_ElasticMoveVel_AcpTrak_0.Deceleration   := Acc_OUT;
	MC_BR_ElasticMoveVel_AcpTrak_0.Jerk           := 0.0;
	MC_BR_ElasticMoveVel_AcpTrak_0.Direction	  := mcDIR_POSITIVE;
	MC_BR_ElasticMoveVel_AcpTrak_0.BufferMode     := mcABORTING;
	MC_BR_ElasticMoveVel_AcpTrak_0();
	MC_BR_ElasticMoveVel_AcpTrak_0.Execute := FALSE;
	// MC_BR_ElasticMoveVel_AcpTrak_1
	MC_BR_ElasticMoveVel_AcpTrak_1.Velocity       := Speed_OUT;
	MC_BR_ElasticMoveVel_AcpTrak_1.Acceleration   := Acc_OUT;
	MC_BR_ElasticMoveVel_AcpTrak_1.Deceleration   := Acc_OUT;
	MC_BR_ElasticMoveVel_AcpTrak_1.Jerk           := 0.0;
	MC_BR_ElasticMoveVel_AcpTrak_1.Direction	  := mcDIR_POSITIVE;
	MC_BR_ElasticMoveVel_AcpTrak_1.BufferMode     := mcABORTING;
	MC_BR_ElasticMoveVel_AcpTrak_1();
	MC_BR_ElasticMoveVel_AcpTrak_1.Execute := FALSE;
	// MC_BR_ElasticMoveVel_AcpTrak_2
	MC_BR_ElasticMoveVel_AcpTrak_2.Velocity       := Speed_OUT;
	MC_BR_ElasticMoveVel_AcpTrak_2.Acceleration   := Acc_OUT;
	MC_BR_ElasticMoveVel_AcpTrak_2.Deceleration   := Acc_OUT;
	MC_BR_ElasticMoveVel_AcpTrak_2.Jerk           := 0.0;
	MC_BR_ElasticMoveVel_AcpTrak_2.Direction	  := mcDIR_POSITIVE;
	MC_BR_ElasticMoveVel_AcpTrak_2.BufferMode     := mcABORTING;
	MC_BR_ElasticMoveVel_AcpTrak_2();
	MC_BR_ElasticMoveVel_AcpTrak_2.Execute := FALSE;
	// MC_ReadStatus
	MC_ReadStatus_0();
	MC_ReadStatus_1();
	MC_ReadStatus_2();

END_PROGRAM
```

### Program Logical/Source/Infrastructure/TrakProduction (IEC) - trak assembly production control

#### Variables.var
```iecst
(*sequence control*)
VAR
	i : USINT; (*FOR LOOP index*)
END_VAR
(*internal data*)
VAR
	NumData : USINT; (*Amount of non-zero data of the producted pouches*)
	ProductionData : ARRAY[0..5] OF UINT; (*Stores the production data every 10 seconds*)
	ProductsPerMinute : REAL;
END_VAR
(*FUB*)
VAR
	TON_0 : TON;
	MTDataMean_0 : MTDataMean;
END_VAR
```

#### Main.st
```iecst
(*********************************************************************************
 * Copyright: B&R Industrial Automation GmbH
 * Author:    	B&R ES
 * Created:   	September 22, 2021/9:53 AM
 * Name:		TrakProduction
 * Description:	Template task to calculate the process product per minute outcome.
				The variable gProducedProduct should be increased in the process
				stations were a new product is produced.
 *********************************************************************************)

PROGRAM _INIT

END_PROGRAM

PROGRAM _CYCLIC

	(***** Find how many non-zero values has the array storing the ProductionData  *****)
	NumData := 0;
	FOR i:=0 TO 5 DO
		IF ProductionData[i] > 0 THEN
			NumData := NumData + 1;
		END_IF
	END_FOR

	(***** Store the Produced Pouches in the ProductionData Array *****)
	// Start the timer
	TON_0.IN := TRUE;
	// Fill the Production Data array
	IF ((TON_0.Q) AND (gProducedProduct > 0)) THEN
		IF (NumData < 6) THEN //The array has not been filled yet
			// Regular production data
			FOR i:=0 TO 5 DO
				IF (ProductionData[i] = 0) THEN
					ProductionData[i] := gProducedProduct;
					EXIT;
				END_IF
			END_FOR
		ELSE
			FOR i:=0 TO 4 DO
				ProductionData[i] := ProductionData[i+1];
			END_FOR
			ProductionData[5] := gProducedProduct;
		END_IF
		// Reset the produced pouches indicator
		gProducedProduct 	:= 0;
		// Reset the timer
		TON_0.IN			:= FALSE;
	END_IF

	(***** Check the Products per Minute *****)
	CASE NumData OF

		1: //100%
			ProductsPerMinute := ProductionData[0]*6;
		2: // 70% 30%
			ProductsPerMinute := (ProductionData[0]*0.3 + ProductionData[1]*0.7)*6;
		3: // 60% 30% 10%
			ProductsPerMinute := (ProductionData[0]*0.1 + ProductionData[1]*0.3 + ProductionData[2]*0.6)*6;
		4: // 55% 25% 15% 5%
			ProductsPerMinute := (ProductionData[0]*0.05 + ProductionData[1]*0.15 + ProductionData[2]*0.25 + ProductionData[3]*0.55)*6;
		5: // 55% 25% 15% 3% 2%
			ProductsPerMinute := (ProductionData[0]*0.02 + ProductionData[1]*0.03 + ProductionData[2]*0.15 + ProductionData[3]*0.25 + ProductionData[4]*0.55)*6;
		6: // 45% 25% 15% 10% 3% 2%
			ProductsPerMinute := (ProductionData[0]*0.02 + ProductionData[1]*0.03 + ProductionData[2]*0.1 + ProductionData[3]*0.15 + ProductionData[4]*0.25 + ProductionData[5]*0.45)*6;
	END_CASE

	(* Mean Production calculation *)
	MTDataMean_0.Enable := gTrakAsm.CmdPower;
	MTDataMean_0.In 	:= ProductsPerMinute;
	MTDataMean_0();

	(***** Reset the Production Data when machine stops *****)
	IF (NOT gTrakAsm.CmdPower) THEN
		FOR i:=0 TO 5 DO
			ProductionData[i] := 0;
		END_FOR
		ProductsPerMinute := 0;
	END_IF

	(***** Call the function blocks *****)
	TON_0.PT := T#10s;
	TON_0();

END_PROGRAM

PROGRAM _EXIT

END_PROGRAM
```

### Program Logical/Source/Infrastructure/TrakSvg (IEC) - trak paper widget control

#### Types.typ
```iecst
TYPE
	StepEnum :
		(
		ASM_INIT,
		ASM_GET_SEGMENT,
		SEG_READ_STATUS,
		SEG_READ_STATUS_WAIT,
		READY
		);
END_TYPE
```

#### Variables.var
```iecst
(*sequence control*)
VAR
	i : UINT;
END_VAR
(*internal data*)
VAR
	SvgTransform : STRING[20000];
	SvgAux : STRING[2];
	ToggleVar : BOOL;
	TON_0 : TON;
END_VAR
```

#### Main.st
```iecst
(*********************************************************************************
 * Copyright: B&R Industrial Automation GmbH
 * Author:    	B&R ES
 * Created:   	November 2, 2021/9:53 AM
 * Name:		TrakSvg
 * Version:   	Tested with mappMotion 5.16.0
 * Description:	Template task to calculate the process product per minute outcome
 * Version 1.0: Generate an svgtransform string in order to monitor the current status
				of all the trak segments.
 *********************************************************************************)

PROGRAM _INIT

	// Possible Segment Status (copy to paper widget colorlist property)
	// colorList -> #CCCCCC,#B3FFB3,#FFFFB3,#FF9999
	// 0 -> Disabled 	(#CCCCCC)
	// 1 -> Ready		(#B3FFB3)
	// 2 -> Stopping	(#FFFFB3)
	// 3 -> ErrorStop	(#FF9999)

//	SvgTransform	:= '[{"select":"#Seg_A_1","fill":3}]';

END_PROGRAM

PROGRAM _CYCLIC

	//////////////////////
	// Open svg transform
	IF gTrakAsm.MonitorSegmentsPresent <> 0 THEN
		SvgTransform := '[';
		FOR i := 1 TO gTrakAsm.MonitorSegmentsPresent DO
			// Save index to auxiliar var
			brsitoa(i,ADR(SvgAux));
			//Build SvgTransform
			brsstrcat(ADR(SvgTransform), ADR('{"select":"#Seg_A_'));
			brsstrcat(ADR(SvgTransform), ADR(SvgAux));
			brsstrcat(ADR(SvgTransform), ADR('","fill":'));
			IF gTrakAsm.Segment[i].StatusReady THEN
				IF gTrakAsm.Segment[i].StatusShuttlesInError THEN
					IF ToggleVar THEN
						brsstrcat(ADR(SvgTransform), ADR('1},'));
					ELSE
						brsstrcat(ADR(SvgTransform), ADR('3},'));
					END_IF
				ELSE
					brsstrcat(ADR(SvgTransform), ADR('1},'));
				END_IF
			ELSIF gTrakAsm.Segment[i].StatusStopping THEN
				brsstrcat(ADR(SvgTransform), ADR('2},'));
			ELSIF gTrakAsm.Segment[i].StatusErrorStop THEN
				brsstrcat(ADR(SvgTransform), ADR('3},'));
			ELSE
				brsstrcat(ADR(SvgTransform), ADR('0},'));
			END_IF
		END_FOR
		// Close svg transform
		brsstrcat(ADR(SvgTransform), ADR('{}]'));
	END_IF

	(* Blinking variable *)
	IF TON_0.Q THEN
		TON_0.IN  := FALSE;
		ToggleVar := NOT ToggleVar;
	ELSE
		TON_0.IN  := TRUE;
	END_IF

	TON_0.PT 	:= T#1s;
	TON_0();

END_PROGRAM

PROGRAM _EXIT

END_PROGRAM
```

### Program Logical/Source/Infrastructure/MappCtrl (IEC) - mapp functionality control

#### Main.st
```iecst
PROGRAM _INIT

	MpAlarmXCore_0.MpLink 	:= ADR(gAlarmXCore);
	MpAlarmXCore_0.Enable	:= TRUE;
	MpAlarmXCore_0();

END_PROGRAM

PROGRAM _CYCLIC

	MpAlarmXCore_0();

END_PROGRAM

PROGRAM _EXIT

	MpAlarmXCore_0.Enable := FALSE;
	MpAlarmXCore_0();

END_PROGRAM
```

Listed in the project but not available here: Logical/Source/ProcessMachine/gProcess.typ
